// TIA Portal project "kazan_basinci_olcumu" (V18)

(* hardware
DEVICE "S7-1200 station_1"  S7-1200 Station
   slot 0: "Rack_0"  S7-1200 Rack  Rack  V1.0
   slot 1: "PLC_1"  CPU 1214C AC/DC/Rly  6ES7 214-1BG40-0XB0  V4.6
*)

// ===== PLC "PLC_1"  CPU 1214C AC/DC/Rly =====

VAR_GLOBAL   // PLC tag table "Default tag table"
   "DEPO BOŞ" AT %I0.0 : Bool;
   "DEPO DOLU" AT %I0.1 : Bool;
   "ANALOG GIRIS" AT %IW64 : Word;
   "ISITICI" AT %Q0.0 : Bool;
   "ALARM" AT %Q0.1 : Bool;
   "POMPA MOTORU" AT %Q0.2 : Bool;
   "Tag_1" AT %MW10 : Word;
END_VAR

ORGANIZATION_BLOCK "Main"   // OB1, LAD, ProgramCycle
TITLE = "Main Program Sweep (Cycle)"
{ S7_Optimized_Access := 'TRUE' }
VERSION : 0.1
// UGULAMA 40: Kazan içerisindeki su isiticilarla kaynatilarak su buhari elde edilmektedir. Kazan basincinin degerini ögrenmek için 24 V gerilimle çalisan basinç dönüstürücü kullanilmaktadir.
// Basinç dönüstürücüsünün algilayabilecegi basinç alant 0-200 kPA olup bu degerle orantili
// olarak 0 - 10 V cikis gerilimi vermektedir. 
// - *Kazan basinci 100 kA'nin altina inince Isiticilarin devreye girmesi ve 175 kPA°hk basinç
// degerinin üstüne gikinca Isiticilarin devre dis kalmasi, 190 kA oldugunda da alarm vermesi
// istenmektedir. Ayrica sivi sevive anahtarindan gelen sinyallere göre pompa kazana su basacaktir.
   VAR_INPUT
      Initial_Call : Bool;   // Initial call of this OB
      Remanence : Bool;   // =True, if remanent data are available
   END_VAR
BEGIN

REGION Network 1
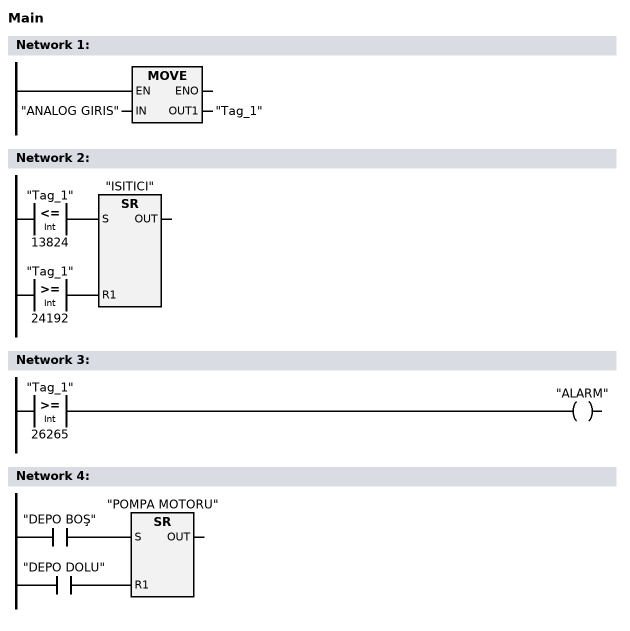
   RUNG wire#powerrail
      Move(in := "ANALOG GIRIS", out1 => "Tag_1")
   END_RUNG
   // the same network as SCL:
   "Tag_1" := "ANALOG GIRIS";
END_REGION

REGION Network 2
   RUNG wire#powerrail
      { S7_Templates := "SrcType := Int" } LE_Contact(in1 := "Tag_1", in2 := 13824)
      S_SR(operand := "ISITICI", r1 := wire#w1)
   END_RUNG
   RUNG wire#powerrail
      { S7_Templates := "SrcType := Int" } GE_Contact(in1 := "Tag_1", in2 := 24192)
   END_RUNG wire#w1
   // the same network as SCL:
   IF "Tag_1" <= 13824 THEN
       "ISITICI" := TRUE;   // SR flip-flop
   END_IF;
   IF "Tag_1" >= 24192 THEN "ISITICI" := FALSE; END_IF;
END_REGION

REGION Network 3
   RUNG wire#powerrail
      { S7_Templates := "SrcType := Int" } GE_Contact(in1 := "Tag_1", in2 := 26265)
      Coil( "ALARM" )
   END_RUNG
   // the same network as SCL:
   "ALARM" := "Tag_1" >= 26265;
END_REGION

REGION Network 4
   RUNG wire#powerrail
      Contact( "DEPO BOŞ" )
      S_SR(operand := "POMPA MOTORU", r1 := wire#w1)
   END_RUNG
   RUNG wire#powerrail
      Contact( "DEPO DOLU" )
   END_RUNG wire#w1
   // the same network as SCL:
   IF "DEPO BOŞ" THEN
       "POMPA MOTORU" := TRUE;   // SR flip-flop
   END_IF;
   IF "DEPO DOLU" THEN "POMPA MOTORU" := FALSE; END_IF;
END_REGION
END_ORGANIZATION_BLOCK